# EPICS autosave request: iocBoot/sioc-b084-bl03/blen_manual.req
file "manual.req" AREA=B084,POS=359,INST=BZ11359A
file "manual.req" AREA=B084,POS=359,INST=BZ11359B
